FUNCTION_BLOCK FB_FastGateValveMonitor
VAR_INPUT
	Closed : BOOL;
	Open : BOOL;
END_VAR
VAR_OUTPUT
	Interlock : BOOL; // MPS shutter
END_VAR
VAR
END_VAR

//Fast acting gate valve - The gate valve will get its instructions from the pressure monitoring, the MPS will only monitor

Interlock := Open AND NOT Closed;

METHOD Control : BOOL
VAR_IN_OUT
	structure : ST_FastGateValveMonitor;
END_VAR
structure.ClosedSt:=Closed;
structure.OpenSt:=Open;
structure.InterlockSt:=Interlock;
END_METHOD

END_FUNCTION_BLOCK

(* stored: Version 1.1.0.1, ProductVersion 3.1.4024.12
   POU FB_FastGateValveMonitor: Id {f82cf651-a3e6-45ef-bb4c-75d6a05fbdb0}, SpecialFunc None
   Method Control: Id {59485de2-f841-4986-948b-d2329e7b50ec} *)
